FUNCTION F_PathCdriveSelectedFile : STRING
VAR_INPUT
	sSelectedPath : STRING(170);
	sSelectedFile : STRING(70);
		
END_VAR
VAR
	sTempSelectedFile : STRING(70);
END_VAR

VAR CONSTANT
	sSlash : STRING(1) := '/';
	sCdrive : STRING(3) := 'C:\';
END_VAR

sSelectedPath := CONCAT(sCdrive,sSelectedPath);
sTempSelectedFile := F_SubStringSelectedFile(sSelectedFile);

(* Generate Path *)
MEMSET(ADR(F_PathCdriveSelectedFile),0,SIZEOF(F_PathCdriveSelectedFile));
MEMCPY(ADR(F_PathCdriveSelectedFile),ADR(sSelectedPath),LEN(sSelectedPath));
MEMCPY(ADR(F_PathCdriveSelectedFile) + LEN(sSelectedPath),ADR(sSlash),LEN(sSlash));
MEMCPY(ADR(F_PathCdriveSelectedFile)+ LEN(sSelectedPath) + LEN(sSlash) ,ADR(sTempSelectedFile) ,LEN(sTempSelectedFile));

END_FUNCTION

(* stored: Version 1.1.0.1, ProductVersion 3.1.4024.6
   POU F_PathCdriveSelectedFile: Id {bd5b36af-fc21-49b0-bfcb-3d786adb7d25}, SpecialFunc None *)
